{attribute 'GeneratedUsingTerminal: IODEVICETYPE_ETHERCATPROT'}
{attribute addProperty BoxType "IODEVICETYPE_ETHERCATPROT"}
{attribute addProperty Id "Beckhoff_EK11xxBeckhoff_EK11xx_811529C670Beckhoff_EK12xxBeckhoff_EK12xx_B10606C62Beckhoff_EK13xxBeckhoff_EK13xx_7663BCA820Beckhoff_EK15xxBeckhoff_EK15xx_47CB6E2F96Beckhoff_EK18xxBeckhoff_EK18xx_88ED272B179Beckhoff_EKM1xxxBeckhoff_EKM1xxx_1191B5D2372Beckhoff_EKx9xxBeckhoff_EKx9xx_85ED516D1090Beckhoff_EKxxxx_0080Beckhoff_EKxxxx_0080_9DDEF9258SyncUnitsSyncUnits_99E584AF18InputsInputs_25A0042B160OutputsOutputs_2397A10E106InfoDataInfoData_C76BEFB322"}
{attribute addProperty CRC "4523609"}
{attribute addProperty Size "2143"}
TYPE EtherCAT_Master_EKxxxx_00450659 :
STRUCT
	{attribute addProperty Name "Beckhoff_EK11xx"}
	{attribute addProperty PreviousPort "EtherCAT_Master_EKxxxx : Master"}
	Beckhoff_EK11xx : Beckhoff_EK11xx_811529C6;
	{attribute addProperty Name "Beckhoff_EK12xx"}
	{attribute addProperty PreviousPort "A_0014(EK1110-0000-0000) : B"}
	Beckhoff_EK12xx : Beckhoff_EK12xx_B10606C6;
	{attribute addProperty Name "Beckhoff_EK13xx"}
	{attribute addProperty PreviousPort "Beckhoff EK12xx : C"}
	Beckhoff_EK13xx : Beckhoff_EK13xx_7663BCA8;
	{attribute addProperty Name "Beckhoff_EK15xx"}
	{attribute addProperty PreviousPort "A_0002(EK1310-0000-0017) : B"}
	Beckhoff_EK15xx : Beckhoff_EK15xx_47CB6E2F;
	{attribute addProperty Name "Beckhoff_EK18xx"}
	{attribute addProperty PreviousPort "Beckhoff EK15xx : C"}
	Beckhoff_EK18xx : Beckhoff_EK18xx_88ED272B;
	{attribute addProperty Name "Beckhoff_EKM1xxx"}
	{attribute addProperty PreviousPort "Beckhoff EK18xx : C"}
	Beckhoff_EKM1xxx : Beckhoff_EKM1xxx_1191B5D2;
	{attribute addProperty Name "Beckhoff_EKx9xx"}
	{attribute addProperty PreviousPort "Beckhoff EKM1xxx : C"}
	Beckhoff_EKx9xx : Beckhoff_EKx9xx_85ED516D;
	{attribute addProperty Name "Beckhoff_EKxxxx_0080"}
	{attribute addProperty PreviousPort "Beckhoff EKx9xx : C"}
	Beckhoff_EKxxxx_0080 : Beckhoff_EKxxxx_0080_9DDEF925;
	{attribute addProperty Name "SyncUnits"}
	SyncUnits : SyncUnits_99E584AF;
	{attribute addProperty Name "Inputs"}
	Inputs : Inputs_25A0042B;
	{attribute addProperty Name "Outputs"}
	Outputs : Outputs_2397A10E;
	{attribute addProperty Name "InfoData"}
	InfoData : InfoData_C76BEFB3;
END_STRUCT
END_TYPE

(* stored: Version 1.2.0.0, ProductVersion 3.1.4024.9
   DUT EtherCAT_Master_EKxxxx_00450659: Id {52a3b904-d172-4d07-a46d-bf2c45905b6e} *)
